FUNCTION_BLOCK FB_CRYO_EVAC_MICADO EXTENDS FB_CRYO_EVAC_BASE_50000
VAR_INPUT
END_VAR
VAR_OUTPUT
END_VAR
VAR
	// Specify pumps
	rp:	FB_CRYO_PUMP_ECODRY;	// Roughing Pump
	tp:	FB_CRYO_PUMP_ATH2303M;	// Turbomolecular Pump
	
END_VAR

SUPER^();	// Execute base FB code.

METHOD M_Configure
VAR_INPUT
END_VAR
//
// Specific MICADO configuration.
//
IF NOT stat.bConfigured	THEN
	//
	// MANDATORY !!!
	// Call base FB::M_Configure() to set the pointers.
	//
	SUPER^.M_Configure();
	

	// MANDATORY: Set References for pumps!!!
	// If not done, system will crash !!!
	rpRef	REF=rp;
	tpRef	REF=tp;
	

	// Specific instance configuration, e.g. anything different
	// from the default values given in the cfg structure of type T_CRYO_EVAC_CFG_50000.
	cfg.nType_VAG1	:= E_CRYO_SENSOR_TYPE_PRESS.WRG_D_NW25;
	cfg.nType_VAG2	:= E_CRYO_SENSOR_TYPE_PRESS.WRG_D_NW25;
	cfg.nType_VAG3	:= E_CRYO_SENSOR_TYPE_PRESS.WRG_D_NW25;
	cfg.nType_VAGF1	:= E_CRYO_SENSOR_TYPE_PRESS.PKR_250;
	cfg.nType_VAGF2	:= E_CRYO_SENSOR_TYPE_PRESS.PKR_250;
	cfg.nType_VAGG1	:= E_CRYO_SENSOR_TYPE_PRESS.PKR_250;
	cfg.nType_VAGG2	:= E_CRYO_SENSOR_TYPE_PRESS.PKR_250;


	stat.bConfigured	:= TRUE;
ELSE
	RETURN;	// Nothing to do any more
END_IF
END_METHOD

METHOD M_ExecuteControllers
VAR_INPUT
END_VAR
//
// Specific MICADO Evacuation System HW configuration.
//

// Roughing Pump	
rp(	
	in_bSimulation	:= FALSE,
	in_sName		:= 'ECODRY V01',
	in_bEnable		:= ctrl.bEnable_PVP,
	in_nSlaveID		:= 31,
	in_sVersion		:= 'V01',
	in_nPeriod		:= 2000);

// Turbo Molecular Pump
tp(	
	in_bSimulation	:= FALSE,
	in_sName		:= 'ATH2303M',
	in_bEnable		:= ctrl.bEnable_TMP,
	in_nModel		:= 2303,
	in_bAutoMonitor	:= TRUE,
	in_nPeriod		:= 2000);

// Valves are controlled in the base FB
SUPER^.M_ExecuteControllers();
END_METHOD

END_FUNCTION_BLOCK

(* stored: Version 1.1.0.1, ProductVersion 3.1.4024.10
   POU FB_CRYO_EVAC_MICADO: Id {a99483db-df13-47b7-aaaa-34ce518a2c72}, SpecialFunc None
   Method M_Configure: Id {e240d503-1f81-4324-a054-3f25dad37d90}
   Method M_ExecuteControllers: Id {e878eb99-7991-4d49-a3ed-85ab05c10992} *)
